TYPE StatusColor :
STRUCT
    fg : Colors; // foreground
    bg : Colors; // background
END_STRUCT
END_TYPE

(* stored: Version 1.1.0.1, ProductVersion 3.1.4018.2
   DUT StatusColor: Id {8430d4fd-9c5b-4a8b-b4b7-e7884df68b92} *)
